FUNCTION_BLOCK ORCHESTRATOR
  {SET_ATTRIBUTE(OpcUa, POINT.STARTPOINT)}
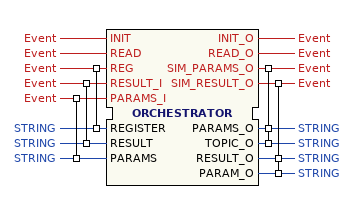
  EVENT_INPUT
    INIT;
    READ;
    REG WITH REGISTER;
    RESULT_I WITH RESULT;
    PARAMS_I WITH PARAMS;
  END_EVENT
  EVENT_OUTPUT
    INIT_O;
    READ_O;
    SIM_PARAMS_O WITH PARAMS_O, TOPIC_O;
    SIM_RESULT_O WITH RESULT_O, PARAM_O;
  END_EVENT
  VAR_INPUT
    REGISTER : STRING; {SET_ATTRIBUTE(OpcUa, Variable)}
    RESULT : STRING; {SET_ATTRIBUTE(OpcUa, Variable)}
    PARAMS : STRING; {SET_ATTRIBUTE(OpcUa, Variable)}
  END_VAR
  VAR_OUTPUT
    PARAMS_O : STRING; {SET_ATTRIBUTE(OpcUa, Variable)}
    TOPIC_O : STRING; {SET_ATTRIBUTE(OpcUa, Variable)}
    RESULT_O : STRING; {SET_ATTRIBUTE(OpcUa, Variable)}
    PARAM_O : STRING; {SET_ATTRIBUTE(OpcUa, Variable)}
  END_VAR
END_FUNCTION_BLOCK
